// TIA Portal V18 export
DATA_BLOCK "gDb_AndonBoxConfig"   // DB17
{ S7_Optimized_Access := 'TRUE' }
VERSION : 0.1
// stored: AutoNumber true, DBAccessibleFromOPCUA true, DBAccessibleFromWebserver true, IsOnlyStoredInLoadMemory false, IsRetainMemResEnabled false, IsWriteProtectedInAS false, MemoryReserve 100
   VAR RETAIN
      flashingPeriod : Time := T#200ms;
      EnableAndon1 : Bool := true;
      EnableAndon2 : Bool := true;
      EnableAndon3 : Bool := true;
      EnableAndon4 : Bool := true;
      EnableAndon5 : Bool := true;
      EnableAndon6 : Bool := true;
      EnableAndon7 : Bool := true;
      EnableAndon8 : Bool;
      EnableAndon9 : Bool;
      EnableAndon10 : Bool;
   END_VAR
BEGIN
END_DATA_BLOCK
